FUNCTION_BLOCK E_PERMITC (* Permissive propagation of an event *)
  (* Standard: 61499-1-A.1 *)
  (* Version 0.3, 2016-04-19, JHC, Holobloc Inc, Corrected spelling of Holobloc. *)
  (* Version 0.2, 2009-11-14, JHC, Holobloci Inc, Updated for 61499-1 2nd Edition. *)
  (* Version 0.1, 2003-12-30, JHC, Rockwell Automation, Updated for 61499-1 CDV. *)
  (* Version 0.0, 2001-03-03, JHC, Rockwell Automation *)
  (* Compiler header: package fb.rt.events; *)
  (* Compiler Java IBM VisualAge 3.0 *)
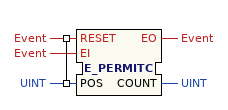
  EVENT_INPUT
    RESET WITH POS; (* Event input *)
    EI;
  END_EVENT
  EVENT_OUTPUT
    EO; (* Event output *)
  END_EVENT
  VAR_INPUT
    POS : UINT; (* Permits EI=>EO pass-through *)
  END_VAR
  VAR_OUTPUT
    COUNT : UINT;
  END_VAR
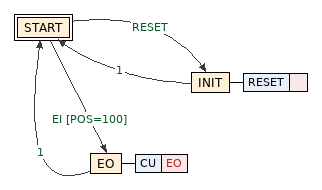
  EC_STATES
    START; (* Initial State *)
    EO : CU -> EO; (* Issue EO Event *)
    INIT : RESET;
  END_STATES
  EC_TRANSITIONS
    EO TO START := 1;
    START TO EO := EI [POS=100];
    START TO INIT := RESET;
    INIT TO START := 1;
  END_TRANSITIONS
  ALGORITHM CU IN ST:
IF POS=100 THEN
	COUNT:=COUNT+1;
END_IF;
  END_ALGORITHM
  ALGORITHM RESET IN ST:
COUNT:=0;
  END_ALGORITHM
END_FUNCTION_BLOCK
